         // Done, Aborted or Error ?
         IF (_response.State >= CmdMessageState.DONE )
         THEN
           // Rest Busy flag
           Busy := FALSE;
           // Update results
           OutCmd.LoadData          := _response.LoadData;
           OutCmd.LoadDataAvailable := _response.LoadDataAvailable;
           // set timeout
           SetTimeout(PT := _timeoutCmd, rTimer := _timerCmd);
           // inc step counter
          _stepCmd := _stepCmd + 1; 
         END_IF
       END_IF


  02: IF ( NOT Execute)
      THEN
        Reset();
      END_IF     

ELSE
  // invalid step
  ErrorID := RobotLibraryEvents.ERR_INVALID_STEP;
END_CASE


// Reset FB
IF ( NOT Execute )
THEN
  Reset();  
END_IF
END_METHOD

METHOD INTERNAL ParseResponsePayload : DINT
VAR_INPUT
  /// Response data
  ResponseData : RobotLibraryRecvDataFB;
  /// Timestamp
  Timestamp    : SystemTime;  
END_VAR
// Table 6-785: Received CMD payload (RC to PLC) of "LoadMeasurementSequential"
// --------------------------
// Header
// --------------------------
// Byte 00 : USINT - ParSeq | State     
// Byte 01 : SINT  - AlarmMessageSeverity    
// Byte 02 : UINT  - AlarmMessageCode HB
// Byte 03 :       - AlarmMessageCode LB
// Datablock
// --------------------------
// Byte 004 : IEC_DATE   - IEC Date LW HB
// Byte 005 :            - IEC Date LW LB
// Byte 006 : IEC_TIME   - IEC Time HW HB
// Byte 007 :            - IEC Time HW LB
// Byte 008 :            - IEC Time LW HB
// Byte 009 :            - IEC Time LW LB
// Byte 010 : REAL       - LoadData.X HW HB
// Byte 011 :            - LoadData.X HW LB
// Byte 012 :            - LoadData.X LW HB
// Byte 013 :            - LoadData.X LW LB
// Byte 014 : REAL       - LoadData.Y HW HB
// Byte 015 :            - LoadData.Y HW LB
// Byte 016 :            - LoadData.Y LW HB
// Byte 017 :            - LoadData.Y LW LB
// Byte 018 : REAL       - LoadData.Z HW HB
// Byte 019 :            - LoadData.Z HW LB
// Byte 020 :            - LoadData.Z LW HB
// Byte 021 :            - LoadData.Z LW LB
// Byte 022 : REAL       - LoadData.Rx HW HB
// Byte 023 :            - LoadData.Rx HW LB
// Byte 024 :            - LoadData.Rx LW HB
// Byte 025 :            - LoadData.Rx LW LB
// Byte 026 : REAL       - LoadData.Ry HW HB
// Byte 027 :            - LoadData.Ry HW LB
// Byte 028 :            - LoadData.Ry LW HB
// Byte 029 :            - LoadData.Ry LW LB
// Byte 030 : REAL       - LoadData.Rz HW HB
// Byte 031 :            - LoadData.Rz HW LB
// Byte 032 :            - LoadData.Rz LW HB
// Byte 033 :            - LoadData.Rz LW LB
// Byte 034 : REAL       - Mass HW HB
// Byte 035 :            - Mass HW LB
// Byte 036 :            - Mass LW HB
// Byte 037 :            - Mass LW LB
// Byte 038 : REAL       - LoadData.Ix HW HB
// Byte 039 :            - LoadData.Ix HW LB
// Byte 040 :            - LoadData.Ix LW HB
// Byte 041 :            - LoadData.Ix LW LB
// Byte 042 : REAL       - LoadData.Iy HW HB
// Byte 043 :            - LoadData.Iy HW LB
// Byte 044 :            - LoadData.Iy LW HB
// Byte 045 :            - LoadData.Iy LW LB
// Byte 046 : REAL       - LoadData.Iz HW HB
// Byte 047 :            - LoadData.Iz HW LB
// Byte 048 :            - LoadData.Iz LW HB
// Byte 049 :            - LoadData.Iz LW LB
// Byte 050 : BOOL       - LoadData.Available
// call base implementation to parse the header from payload buffer
ResponseData.PayloadPtr := SUPER^.ParseResponsePayload(ResponseData := ResponseData, Timestamp := Timestamp);

// copy parsed header to response
_response.ParSeq               := _rspHeader.ParSeq;
_response.State                := _rspHeader.State;
_response.AlarmMessageSeverity := _rspHeader.AlarmMessageSeverity;
_response.AlarmMessageCode     := _rspHeader.AlarmMessageCode;

// Get Response.LoadData.Timestamp.TsData
_response.LoadData.Timestamp.IEC_DATE := ResponseData.GetIecDate();
// Get Response.LoadData.Timestamp.TsTime
_response.LoadData.Timestamp.IEC_TIME := ResponseData.GetIecTime();
// Get Response.LoadData.X
_response.LoadData.X := ResponseData.GetReal();
// Get Response.LoadData.Y
_response.LoadData.Y := ResponseData.GetReal();
// Get Response.LoadData.Z
_response.LoadData.Z := ResponseData.GetReal();
// Get Response.LoadData.Rx
_response.LoadData.Rx := ResponseData.GetReal();
// Get Response.LoadData.Ry
_response.LoadData.Ry := ResponseData.GetReal();
// Get Response.LoadData.Rz
_response.LoadData.Rz := ResponseData.GetReal();
// Get Response.LoadData.Mass
_response.LoadData.Mass := ResponseData.GetReal();
// Get Response.LoadData.Ix
_response.LoadData.Ix := ResponseData.GetReal();
// Get Response.LoadData.Iy
_response.LoadData.Iy := ResponseData.GetReal();
// Get Response.LoadData.Iz
_response.LoadData.Iz := ResponseData.GetReal();
// Get Response.LoadDataAvailable
_response.LoadDataAvailable := ResponseData.GetBool();

// Create logging
ParseResponsePayloadLog(ResponseData := ResponseData, Timestamp := Timestamp);
END_METHOD

METHOD INTERNAL ParseResponsePayloadLog
VAR_INPUT
  /// Response data
  ResponseData : RobotLibraryRecvDataFB;
  /// Timestamp
  Timestamp    : SystemTime;  
END_VAR
// Create log entry for Parameter start
CreateLogMessage      ( Timestamp   := Timestamp,
                        MessageType := MessageType.CMD,
                        Severity    := Severity.DEBUG,
                        MessageCode := 0,
                        MessageText := 'Parsed the following parameter(s) from response data:');
                        
// Create log entry for LoadData.Timestamp.IEC_DATE
CreateLogMessagePara1 ( Timestamp   := Timestamp,
                        MessageType := MessageType.CMD,
                        Severity    := Severity.DEBUG,
                        MessageCode := 0,
                        MessageText := 'Response.LoadData.Timestamp.IEC_DATE = {1}',
                        Para1       :=  IEC_DATE_TO_STRING(_response.LoadData.Timestamp.IEC_DATE));

// Create log entry for LoadData.Timestamp.IEC_TIME
CreateLogMessagePara1 ( Timestamp   := Timestamp,
                        MessageType := MessageType.CMD,
                        Severity    := Severity.DEBUG,
                        MessageCode := 0,
                        MessageText := 'Response.LoadData.Timestamp.IEC_TIME = {1}',
                        Para1       :=  IEC_TIME_TO_STRING(_response.LoadData.Timestamp.IEC_TIME));

// Create log entry for LoadData.X
CreateLogMessagePara1 ( Timestamp   := Timestamp,
                        MessageType := MessageType.CMD,
                        Severity    := Severity.DEBUG,
                        MessageCode := 0,
                        MessageText := 'Response.LoadData.X = {1}',
                        Para1       :=  REAL_TO_STRING(_response.LoadData.X));

// Create log entry for LoadData.Y
CreateLogMessagePara1 ( Timestamp   := Timestamp,
                        MessageType := MessageType.CMD,
                        Severity    := Severity.DEBUG,
                        MessageCode := 0,
                        MessageText := 'Response.LoadData.Y = {1}',
                        Para1       :=  REAL_TO_STRING(_response.LoadData.Y));

// Create log entry for LoadData.Z
CreateLogMessagePara1 ( Timestamp   := Timestamp,
                        MessageType := MessageType.CMD,
                        Severity    := Severity.DEBUG,
                        MessageCode := 0,
                        MessageText := 'Response.LoadData.Z = {1}',
                        Para1       :=  REAL_TO_STRING(_response.LoadData.Z));

// Create log entry for LoadData.Rx
CreateLogMessagePara1 ( Timestamp   := Timestamp,
                        MessageType := MessageType.CMD,
                        Severity    := Severity.DEBUG,
                        MessageCode := 0,
                        MessageText := 'Response.LoadData.Rx = {1}',
                        Para1       :=  REAL_TO_STRING(_response.LoadData.Rx));

// Create log entry for LoadData.Ry
CreateLogMessagePara1 ( Timestamp   := Timestamp,
                        MessageType := MessageType.CMD,
                        Severity    := Severity.DEBUG,
                        MessageCode := 0,
                        MessageText := 'Response.LoadData.Ry = {1}',
                        Para1       :=  REAL_TO_STRING(_response.LoadData.Ry));

// Create log entry for LoadData.Rz
CreateLogMessagePara1 ( Timestamp   := Timestamp,
                        MessageType := MessageType.CMD,
                        Severity    := Severity.DEBUG,
                        MessageCode := 0,
                        MessageText := 'Response.LoadData.Rz = {1}',
                        Para1       :=  REAL_TO_STRING(_response.LoadData.Rz));

// Create log entry for LoadData.Mass
CreateLogMessagePara1 ( Timestamp   := Timestamp,
                        MessageType := MessageType.CMD,
                        Severity    := Severity.DEBUG,
                        MessageCode := 0,
                        MessageText := 'Response.LoadData.Mass = {1}',
                        Para1       :=  REAL_TO_STRING(_response.LoadData.Mass));

// Create log entry for LoadData.Ix
CreateLogMessagePara1 ( Timestamp   := Timestamp,
                        MessageType := MessageType.CMD,
                        Severity    := Severity.DEBUG,
                        MessageCode := 0,
                        MessageText := 'Response.LoadData.Ix = {1}',
                        Para1       :=  REAL_TO_STRING(_response.LoadData.Ix));

// Create log entry for LoadData.Iy
CreateLogMessagePara1 ( Timestamp   := Timestamp,
                        MessageType := MessageType.CMD,
                        Severity    := Severity.DEBUG,
                        MessageCode := 0,
                        MessageText := 'Response.LoadData.Iy = {1}',
                        Para1       :=  REAL_TO_STRING(_response.LoadData.Iy));

// Create log entry for LoadData.Iz
CreateLogMessagePara1 ( Timestamp   := Timestamp,
                        MessageType := MessageType.CMD,
                        Severity    := Severity.DEBUG,
                        MessageCode := 0,
                        MessageText := 'Response.LoadData.Iz = {1}',
                        Para1       :=  REAL_TO_STRING(_response.LoadData.Iz));

// Create log entry for LoadDataAvailable
CreateLogMessagePara1 ( Timestamp   := Timestamp,
                        MessageType := MessageType.CMD,
                        Severity    := Severity.DEBUG,
                        MessageCode := 0,
                        MessageText := 'Response.LoadDataAvailable = {1}',
                        Para1       :=  BOOL_TO_STRING(_response.LoadDataAvailable));
END_METHOD

METHOD PROTECTED Reset : DINT
VAR_INPUT
END_VAR
Reset := SUPER^.Reset();

Done               := FALSE;
Busy               := FALSE;
Active             := FALSE;
CommandBuffered    := FALSE;
CommandAborted     := FALSE;
CommandInterrupted := FALSE;
END_METHOD

END_FUNCTION_BLOCK

// Library/POUs/ConveyorTracking/MC_ActivateConveyorTracking/MC_ActivateConveyorTrackingFB
/// Activate conveyor tracking mode
FUNCTION_BLOCK MC_ActivateConveyorTrackingFB EXTENDS RobotLibraryBaseFB
// ------------------------------------------------------------------------- 
//  SRCI Robot Library                                                
// ------------------------------------------------------------------------- 
//                                                                           
//  Object:      ActivateConveyorTrackingFB                                       
//  Author:      Thorsten Brach                                                
//  Date:        2024-06-11
//
//  Description:                                              
//   
//                                                                           
//  Copyright: 
//    (C) 2024 Thorsten Brach. All rights reserved                                                                                                                                            
//             Licensed under the LGPL-3.0 license.
//                                                                           
//  Disclaimer:                                                                           
//    This project is provided without any guarantee and can be used for   
//    private and commercial purposes. Any use is at the user’s 
//    own risk and responsibility.
//
// -------------------------------------------------------------------------
VAR_INPUT
  /// SSet TRUE to activate conveyor tracking functionality
  Enable             : BOOL;
  /// Command parameter 
  ParCmd             : ActivateConveyorTrackingParCmd;      
END_VAR

VAR_OUTPUT
  /// TRUE, while the following outputs return valid values:
  /// • TrackingStatusByte
  /// • RCEncoderValue
  Valid              : BOOL;
  /// FB is being processed
  Busy               : BOOL;
  /// Command is transferred and confirmed by the RC
  CommandBuffered    : BOOL;
  /// Receiving of input parameter values has been acknowledged by RC
  ParameterAccepted  : BOOL;
  /// Command output 
  OutCmd             : ActivateConveyorTrackingOutCmd;  
END_VAR

VAR
  /// internal copy of command parameter 
 _parCmd             : ActivateConveyorTrackingParCmd;
  /// command data to send
 _command            : ActivateConveyorTrackingSendData;
  /// response data received
 _response           : ActivateConveyorTrackingRecvData;  
  /// Rising edge for enable
 _enable_R          : R_TRIG;
  /// Falling edge for enable
 _enable_F          : F_TRIG;    
END_VAR

SUPER^(AxesGroup := AxesGroup);

METHOD PROTECTED CheckFunctionSupported : BOOL
VAR_IN_OUT
  /// Robot assignment of function
  AxesGroup : AxesGroup; 
END_VAR
CheckFunctionSupported := AxesGroup.InternalData.RCSupportedFunctions.ActivateConveyorTracking;

IF ( NOT CheckFunctionSupported )
THEN
  // call base implementation for set error and create log entry
  SUPER^.CheckFunctionSupported(AxesGroup := AxesGroup);
END_IF
END_METHOD

METHOD PROTECTED CheckParameterChanged : BOOL
VAR_IN_OUT
  /// Robot assignment of function
  AxesGroup    : AxesGroup; 
END_VAR
// Check ParCmd Size is > 0, because MemCmp does not work correctly with size = 0
IF (SIZEOF(ParCmd) = 0) 
THEN 
  RETURN;
END_IF

// compare memory 
_parameterChanged := ( SysDepMemCmp(pData1 := ADR(ParCmd), pData2 := ADR(_parCmd), DataLen := SIZEOF(ParCmd)) <> RobotLibraryConstants.OK );

// check parameter valid ?
_parameterValid   := CheckParameterValid( AxesGroup := AxesGroup );

IF ((  _parameterChanged        )  AND 
    (  _parameterValid          )) OR
    (  _parameterUpdateInternal )  
THEN  
  // reset internal flag for send parameter update
 _parameterUpdateInternal := FALSE;
  // update internal copy of parameters 
 _parCmd := ParCmd;
  // inc parameter sequence
 _command.ParSeq := _command.ParSeq + 1;
  // update command data  
  CommandData := CreateCommandPayload(AxesGroup := AxesGroup); // ( Access via reference to rCommandFB in ACR )
  // notify active command register 
  AxesGroup.Acyclic.ActiveCommandRegister.NotifyParameterChanged := _uniqueID;
  // Reset parameter accepted flag
  ParameterAccepted := FALSE;  
END_IF
END_METHOD

METHOD INTERNAL CreateCommandPayload : RobotLibrarySendDataFB
VAR_IN_OUT
  /// Robot assignment of function
  AxesGroup : AxesGroup; 
END_VAR
// Table 6-438: Sent CMD payload (PLC to RC) of "ActivateConveyorTracking"
// --------------------------
// Header
// --------------------------
// Byte 00 : UINT  - Type HB     
// Byte 01 :       - Type LB    
// Byte 02 : USINT - Reserve | ExecutionMode
// Byte 03 : USINT - ParSeq  | Priority
// --------------------------
// Datablock
// --------------------------
// Byte 04 : SINT  - ConveyorNo
// Byte 05 : SINT  - ConnectionMode
// --------------------------


// set command parameter 
_command.CmdTyp         :=  CmdType.ActivateConveyorTracking;
_command.ExecMode       :=  ExecMode;
_command.ParSeq         := _command.ParSeq;
_command.Priority       :=  Priority;
_command.ConveyorNo     := _parCmd.ConveyorNo;
_command.ConnectionMode := _parCmd.ConnectionMode;


// copy command data to header
_cmdHeader := _command;
// call base implementation to copy header to payload buffer
CreateCommandPayload := SUPER^.CreateCommandPayload(AxesGroup := AxesGroup);


// add command.ConveyorNo
CreateCommandPayload.AddSint(_command.ConveyorNo);
// add command.ConnectionMode
CreateCommandPayload.AddSint(_command.ConnectionMode);

// Create logging
CreateCommandPayloadLog(AxesGroup := AxesGroup);
END_METHOD

METHOD INTERNAL CreateCommandPayloadLog 
VAR_IN_OUT
  /// Robot assignment of function
  AxesGroup : AxesGroup; 
END_VAR
// Create log entry for Parameter start
CreateLogMessage      ( Timestamp   := AxesGroup.InternalData.SystemTime,
                        MessageType := MessageType.CMD,
                        Severity    := Severity.DEBUG,
                        MessageCode := 0,
                        MessageText := 'Create command payload with the following parameter(s) :');

// Create log entry for ConveyorNo
CreateLogMessagePara1 ( Timestamp   := AxesGroup.InternalData.SystemTime,
                        MessageType := MessageType.CMD,
                        Severity    := Severity.DEBUG,
                        MessageCode := 0,
                        MessageText := 'Command.ConveyorNo = {1}',
                        Para1       :=  SINT_TO_STRING(_command.ConveyorNo));
                        
// Create log entry for ConnectionMode
CreateLogMessagePara1 ( Timestamp   := AxesGroup.InternalData.SystemTime,
                        MessageType := MessageType.CMD,
                        Severity    := Severity.DEBUG,
                        MessageCode := 0,
                        MessageText := 'Command.ConnectionMode = {1}',
                        Para1       :=  CONNECTION_MODE_TO_STRING(_command.ConnectionMode));
END_METHOD

METHOD FB_init : BOOL
VAR_INPUT
  /// if TRUE, the retain variables are initialized (warm start / cold start)
  bInitRetains : BOOL; 
  /// if TRUE, the instance afterwards gets moved into the copy code (online change)
  bInCopyCode  : BOOL;  
END_VAR
MyType := 'MC_ActivateConveyorTrackingFB';
END_METHOD

METHOD PROTECTED OnCall
VAR_IN_OUT
  /// Robot assignment of function
  AxesGroup : AxesGroup; 
END_VAR
// call base implementation
SUPER^.OnCall(AxesGroup := AxesGroup);

// building rising and falling edges
_enable_R( CLK := Enable);
_enable_F( CLK := Enable);

CASE _stepCmd OF
  
  00:  IF ( _enable_R.Q ) 
       THEN
         // reset the rising edge
        _enable_R();       
         // reset the falling edge
        _enable_F();       

         // Check function is supported and parameter are valid ?
         IF (( CheckFunctionSupported( AxesGroup := AxesGroup )) AND
             ( CheckParameterValid   ( AxesGroup := AxesGroup )))      
         THEN
           // set busy flag
           Busy := TRUE;
           // Reset command outputs
           SysDepMemSet(pDest := ADR(OutCmd), Value := 0, DataLen := SIZEOF(OutCmd));         
           // apply command parameter
          _parCmd := ParCmd;
           // init parameter sequence
          _command.ParSeq := 1;
           // create command data
           CommandData := CreateCommandPayload(AxesGroup := AxesGroup);
           // Add command to active command register
          _uniqueID := AxesGroup.Acyclic.ActiveCommandRegister.AddCmd( pCommandFB := ADR(THIS^ ));     
           // set timeout
           SetTimeout(PT := _timeoutCmd, rTimer := _timerCmd);
           // inc step counter
          _stepCmd := _stepCmd + 1;
         END_IF 
       END_IF
     

  01:  // Wait for responce received
       IF ( _responseReceived )
       THEN
         // reset response received flag
        _responseReceived := FALSE;

         CASE  _response.State 
         OF
           CmdMessageState.BUFFERED    : CommandBuffered    := TRUE;
           CmdMessageState.ACTIVE      : ParameterAccepted  := TRUE;           
           CmdMessageState.ERROR       : Error              := TRUE;
         END_CASE
                
         // Done, Aborted or Error ?
         IF (_response.State >= CmdMessageState.DONE )
         THEN
           // Update results
           OutCmd.TrackingStatus := _response.TrackingStatus;
           // set timeout
           SetTimeout(PT := _timeoutCmd, rTimer := _timerCmd);
           // inc step counter
          _stepCmd := _stepCmd + 1; 
         END_IF
       END_IF


  02: IF (NOT Enable)
      THEN
        Reset();
	    END_IF
      
ELSE
  // invalid step
  ErrorID := RobotLibraryEvents.ERR_INVALID_STEP;
END_CASE



// Reset FB
IF (( _enable_R.Q ) OR
    ( _enable_F.Q ))
THEN
  Reset();
END_IF
END_METHOD

METHOD INTERNAL ParseResponsePayload : DINT
VAR_INPUT
  /// Response data
  ResponseData : RobotLibraryRecvDataFB;
  /// Timestamp
  Timestamp    : SystemTime;  
END_VAR
// Table 6-439: Received CMD payload (RC to PLC) of "ActivateConveyorTracking"
// --------------------------
// Header
// --------------------------
// Byte 00 : USINT - ParSeq | State     
// Byte 01 : SINT  - AlarmMessageSeverity    
// Byte 02 : UINT  - AlarmMessageCode HB
// Byte 03 :       - AlarmMessageCode LB
// --------------------------
// Datablock
// --------------------------
// Byte 04 : BYTE  - TrackingStatusByte
// --------------------------
// call base implementation to parse the header from payload buffer
ResponseData.PayloadPtr := SUPER^.ParseResponsePayload(ResponseData := ResponseData, Timestamp := Timestamp);

// copy parsed header to response
_response.ParSeq               := _rspHeader.ParSeq;
_response.State                := _rspHeader.State;
_response.AlarmMessageSeverity := _rspHeader.AlarmMessageSeverity;
_response.AlarmMessageCode     := _rspHeader.AlarmMessageCode;

// Get Response.Enabled
_response.TrackingStatus := ResponseData.GetTrackingStatus();

// Create logging
ParseResponsePayloadLog(ResponseData := ResponseData, Timestamp := Timestamp);
END_METHOD

METHOD INTERNAL ParseResponsePayloadLog
VAR_INPUT
  /// Response data
  ResponseData : RobotLibraryRecvDataFB;
  /// Timestamp
  Timestamp    : SystemTime;  
END_VAR
// Create log entry for Parameter start
CreateLogMessage      ( Timestamp   := Timestamp,
                        MessageType := MessageType.CMD,
                        Severity    := Severity.DEBUG,
                        MessageCode := 0,
                        MessageText := 'Parsed the following parameter(s) from response data:');
                        
// Create log entry for TrackingStatus.ConveyorTrackingEnabled
CreateLogMessagePara1 ( Timestamp   := Timestamp,
                        MessageType := MessageType.CMD,
                        Severity    := Severity.DEBUG,
                        MessageCode := 0,
                        MessageText := 'Response.TrackingStatus.ConveyorTrackingEnabled = {1}',
                        Para1       :=  BOOL_TO_STRING(_response.TrackingStatus.ConveyorTrackingEnabled));

// Create log entry for TrackingStatus.WaitingForSynchronization
CreateLogMessagePara1 ( Timestamp   := Timestamp,
                        MessageType := MessageType.CMD,
                        Severity    := Severity.DEBUG,
                        MessageCode := 0,
                        MessageText := 'Response.TrackingStatus.WaitingForSynchronization = {1}',
                        Para1       :=  BOOL_TO_STRING(_response.TrackingStatus.WaitingForSynchronization));

// Create log entry for TrackingStatus.Synchronizing
CreateLogMessagePara1 ( Timestamp   := Timestamp,
                        MessageType := MessageType.CMD,
                        Severity    := Severity.DEBUG,
                        MessageCode := 0,
                        MessageText := 'Response.TrackingStatus.Synchronizing = {1}',
                        Para1       :=  BOOL_TO_STRING(_response.TrackingStatus.Synchronizing));

// Create log entry for TrackingStatus.Synchronous
CreateLogMessagePara1 ( Timestamp   := Timestamp,
                        MessageType := MessageType.CMD,
                        Severity    := Severity.DEBUG,
                        MessageCode := 0,
                        MessageText := 'Response.TrackingStatus.Synchronous = {1}',
                        Para1       :=  BOOL_TO_STRING(_response.TrackingStatus.Synchronous));

// Create log entry for TrackingStatus.Desynchronizing
CreateLogMessagePara1 ( Timestamp   := Timestamp,
                        MessageType := MessageType.CMD,
                        Severity    := Severity.DEBUG,
                        MessageCode := 0,
                        MessageText := 'Response.TrackingStatus.Desynchronizing = {1}',
                        Para1       :=  BOOL_TO_STRING(_response.TrackingStatus.Desynchronizing));

// Create log entry for TrackingStatus.SyncOutZoneEntered
CreateLogMessagePara1 ( Timestamp   := Timestamp,
                        MessageType := MessageType.CMD,
                        Severity    := Severity.DEBUG,
                        MessageCode := 0,
                        MessageText := 'Response.TrackingStatus.SyncOutZoneEntered = {1}',
                        Para1       :=  BOOL_TO_STRING(_response.TrackingStatus.SyncOutZoneEntered));

// Create log entry for TrackingStatus.SyncOutZoneLeft
CreateLogMessagePara1 ( Timestamp   := Timestamp,
                        MessageType := MessageType.CMD,
                        Severity    := Severity.DEBUG,
                        MessageCode := 0,
                        MessageText := 'Response.TrackingStatus.SyncOutZoneLeft = {1}',
                        Para1       :=  BOOL_TO_STRING(_response.TrackingStatus.SyncOutZoneLeft));

// Create log entry for TrackingStatus.NotUsed
CreateLogMessagePara1 ( Timestamp   := Timestamp,
                        MessageType := MessageType.CMD,
                        Severity    := Severity.DEBUG,
                        MessageCode := 0,
                        MessageText := 'Response.TrackingStatus.NotUsed = {1}',
                        Para1       :=  BOOL_TO_STRING(_response.TrackingStatus.NotUsed));
END_METHOD

METHOD PROTECTED Reset : DINT
VAR_INPUT
END_VAR
Reset := SUPER^.Reset();

Valid              := FALSE;
Busy               := FALSE;
CommandBuffered    := FALSE;
ParameterAccepted  := FALSE;
END_METHOD

END_FUNCTION_BLOCK

// Library/POUs/ConveyorTracking/MC_ConfigureConveyor/MC_ConfigureConveyorFB
/// Configure conveyor parameters
FUNCTION_BLOCK MC_ConfigureConveyorFB EXTENDS RobotLibraryBaseExecuteFB
// ------------------------------------------------------------------------- 
//  SRCI Robot Library                                                
// ------------------------------------------------------------------------- 
//                                                                           
//  Object:      ConfigureConveyorFB                                       
//  Author:      Thorsten Brach                                                
//  Date:        2024-06-11
//
//  Description:                                              
//   
//                                                                           
//  Copyright: 
//    (C) 2024 Thorsten Brach. All rights reserved                                                                                                                                            
//             Licensed under the LGPL-3.0 license.
//                                                                           
//  Disclaimer:                                                                           
//    This project is provided without any guarantee and can be used for   
//    private and commercial purposes. Any use is at the user’s 
//    own risk and responsibility.
//
// -------------------------------------------------------------------------
VAR_INPUT
  /// Command parameter 
  ParCmd          : ConfigureConveyorParCmd;      
END_VAR

VAR_OUTPUT
  /// Command is transferred and confirmed by the RC
  CommandBuffered : BOOL;
  /// Command output 
  OutCmd          : ConfigureConveyorOutCmd;  
END_VAR

VAR
  /// internal copy of command parameter 
 _parCmd          : ConfigureConveyorParCmd;
  /// command data to send
 _command         : ConfigureConveyorSendData;
  /// response data received
 _response        : ConfigureConveyorRecvData;      
END_VAR

SUPER^(AxesGroup := AxesGroup);

METHOD PROTECTED CheckFunctionSupported : BOOL
VAR_IN_OUT
  /// Robot assignment of function
  AxesGroup : AxesGroup; 
END_VAR
CheckFunctionSupported := AxesGroup.InternalData.RCSupportedFunctions.ConfigureConveyor;

IF ( NOT CheckFunctionSupported )
THEN
  // call base implementation for set error and create log entry
  SUPER^.CheckFunctionSupported(AxesGroup := AxesGroup);
END_IF
END_METHOD

METHOD PROTECTED CheckParameterChanged : BOOL
VAR_IN_OUT
  /// Robot assignment of function
  AxesGroup    : AxesGroup; 
END_VAR
// Check ParCmd Size is > 0, because MemCmp does not work correctly with size = 0
IF (SIZEOF(ParCmd) = 0) 
THEN 
  RETURN;
END_IF

// compare memory 
_parameterChanged := ( SysDepMemCmp(pData1 := ADR(ParCmd), pData2 := ADR(_parCmd), DataLen := SIZEOF(ParCmd)) <> RobotLibraryConstants.OK );

// check parameter valid ?
_parameterValid   := CheckParameterValid( AxesGroup := AxesGroup );

IF ((  _parameterChanged        )  AND 
    (  _parameterValid          )) OR
    (  _parameterUpdateInternal )  
THEN  
  // reset internal flag for send parameter update
 _parameterUpdateInternal := FALSE;
  // update internal copy of parameters 
 _parCmd := ParCmd;
  // inc parameter sequence
 _command.ParSeq := _command.ParSeq + 1;
  // update command data  
  CommandData := CreateCommandPayload(AxesGroup := AxesGroup); // ( Access via reference to rCommandFB in ACR )
  // notify active command register 
  AxesGroup.Acyclic.ActiveCommandRegister.NotifyParameterChanged := _uniqueID;
END_IF
END_METHOD

METHOD INTERNAL CreateCommandPayload : RobotLibrarySendDataFB
VAR_IN_OUT
  /// Robot assignment of function
  AxesGroup : AxesGroup; 
END_VAR
// Table 6-458: Sent CMD payload (PLC to RC) of "ConfigureConveyor"
// --------------------------
// Header
// --------------------------
// Byte 00 : UINT       - Type HB     
// Byte 01 :            - Type LB    
// Byte 02 : USINT      - Reserve | ExecutionMode
// Byte 03 : USINT      - ParSeq  | Priority
// --------------------------
// Datablock
// --------------------------
// Byte 04 : IEC_DATE   - Date              LW HB
// Byte 05 :            - Date              LW LB
// Byte 06 : IEC_TIME   - Time              HW HB
// Byte 07 :            - Time              HW LB
// Byte 08 :            - Time              LW HB
// Byte 09 :            - Time              LW LB
// Byte 10 : USINT      - ReferenceFrame
// Byte 11 : BYTE       - Reserve
// Byte 12 : REAL       - ConveyorOrigin.X  HW HB
// Byte 13 :            - ConveyorOrigin.X  HW LB
// Byte 14 :            - ConveyorOrigin.X  LW HB
// Byte 15 :            - ConveyorOrigin.X  LW LB
// Byte 16 : REAL       - ConveyorOrigin.Y  HW HB
// Byte 17 :            - ConveyorOrigin.Y  HW LB
// Byte 18 :            - ConveyorOrigin.Y  LW HB
// Byte 19 :            - ConveyorOrigin.Y  LW LB
// Byte 20 : REAL       - ConveyorOrigin.Z  HW HB
// Byte 21 :            - ConveyorOrigin.Z  HW LB
// Byte 22 :            - ConveyorOrigin.Z  LW HB
// Byte 23 :            - ConveyorOrigin.Z  LW LB
// Byte 24 : REAL       - ConveyorOrigin.Rx HW HB
// Byte 25 :            - ConveyorOrigin.Rx HW LB
// Byte 26 :            - ConveyorOrigin.Rx LW HB
// Byte 27 :            - ConveyorOrigin.Rx LW LB
// Byte 28 : REAL       - ConveyorOrigin.Ry HW HB
// Byte 29 :            - ConveyorOrigin.Ry HW LB
// Byte 30 :            - ConveyorOrigin.Ry LW HB
// Byte 31 :            - ConveyorOrigin.Ry LW LB
// Byte 32 : REAL       - ConveyorOrigin.Rz HW HB
// Byte 33 :            - ConveyorOrigin.Rz HW LB
// Byte 34 :            - ConveyorOrigin.Rz LW HB
// Byte 35 :            - ConveyorOrigin.Rz LW LB
// Byte 36 : BOOL       - ConveyorOrigin Available
// Byte 37 : USINT      - ConveyorNo
// Byte 38 : USINT      - ConveyorType
// Byte 39 : REAL       - Radius            HW HB
// Byte 40 :            - Radius            HW LB
// Byte 41 :            - Radius            LW HB
// Byte 42 :            - Radius            LW LB
// Byte 43 : REAL       - StartDistance     HW HB
// Byte 44 :            - StartDistance     HW LB
// Byte 45 :            - StartDistance     LW HB
// Byte 46 :            - StartDistance     LW LB
// Byte 47 : REAL       - EndDistance       HW HB
// Byte 48 :            - EndDistance       HW LB
// Byte 49 :            - EndDistance       LW HB
// Byte 50 :            - EndDistance       LW LB
// Byte 51 : REAL       - SyncInLength      HW HB
// Byte 52 :            - SyncInLength      HW LB
// Byte 53 :            - SyncInLength      LW HB
// Byte 54 :            - SyncInLength      LW LB
// Byte 55 : REAL       - SyncOutLength     HW HB
// Byte 56 :            - SyncOutLength     HW LB
// Byte 57 :            - SyncOutLength     LW HB
// Byte 58 :            - SyncOutLength     LW LB
// --------------------------
// set command parameter 
_command.CmdTyp         :=  CmdType.ConfigureConveyor;
_command.ExecMode       :=  ExecMode;
_command.ParSeq         := _command.ParSeq;
_command.Priority       :=  Priority;
_command.ConveyorNo     := _parCmd.ConveyorNo;
_command.ConveyorOrigin := _parCmd.ConveyorOrigin;
_command.ConveyorType   := _parCmd.ConveyorType;
_command.Radius         := _parCmd.Radius;
_command.StartDistance  := _parCmd.StartDistance;
_command.EndDistance    := _parCmd.EndDistance;
_command.SyncInLength   := _parCmd.SyncInLength;
_command.SyncOutLength  := _parCmd.SyncOutLength;

// copy command data to header
_cmdHeader := _command;
// call base implementation to copy header to payload buffer
CreateCommandPayload := SUPER^.CreateCommandPayload(AxesGroup := AxesGroup);


// add command.ConveyorOrigin.Timestamp.IEC_DATE
CreateCommandPayload.AddIecDate(_command.ConveyorOrigin.Timestamp.IEC_DATE);
// add command.ConveyorOrigin.Timestamp.IEC_TIME
CreateCommandPayload.AddIecTime(_command.ConveyorOrigin.Timestamp.IEC_TIME);
// add command.ConveyorOrigin.ReferenceFrame
CreateCommandPayload.AddUsint(_command.ConveyorOrigin.ReferenceFrame);
// add command.ConveyorOrigin.Reserve
CreateCommandPayload.AddByte(0);
// add command.ConveyorOrigin.ReferenceFrame.X
CreateCommandPayload.AddReal(_command.ConveyorOrigin.X);
// add command.ConveyorOrigin.ReferenceFrame.Y
CreateCommandPayload.AddReal(_command.ConveyorOrigin.Y);
// add command.ConveyorOrigin.ReferenceFrame.Z
CreateCommandPayload.AddReal(_command.ConveyorOrigin.Z);
// add command.ConveyorOrigin.ReferenceFrame.Rx
CreateCommandPayload.AddReal(_command.ConveyorOrigin.Rx);
// add command.ConveyorOrigin.ReferenceFrame.Ry
CreateCommandPayload.AddReal(_command.ConveyorOrigin.Ry);
// add command.ConveyorOrigin.ReferenceFrame.Rz
CreateCommandPayload.AddReal(_command.ConveyorOrigin.Rz);
// add command.ConveyorOriginAvailable
CreateCommandPayload.AddBool(_command.ConveyorOriginAvailable);
// add command.ConveyorNo
CreateCommandPayload.AddUsint(_command.ConveyorNo);
// add command.ConveyorType
CreateCommandPayload.AddUsint(_command.ConveyorType);
// add command.Radius
CreateCommandPayload.AddReal(_command.Radius);
// add command.StartDistance
CreateCommandPayload.AddReal(_command.StartDistance);
// add command.EndDistance
CreateCommandPayload.AddReal(_command.EndDistance);
// add command.SyncInLength
CreateCommandPayload.AddReal(_command.SyncInLength);
// add command.SyncOutLength
CreateCommandPayload.AddReal(_command.SyncOutLength);

// Create logging
CreateCommandPayloadLog(AxesGroup := AxesGroup);
END_METHOD

METHOD INTERNAL CreateCommandPayloadLog 
VAR_IN_OUT
  /// Robot assignment of function
  AxesGroup : AxesGroup; 
END_VAR
// Create log entry for Parameter start
CreateLogMessage      ( Timestamp   := AxesGroup.InternalData.SystemTime,
                        MessageType := MessageType.CMD,
                        Severity    := Severity.DEBUG,
                        MessageCode := 0,
                        MessageText := 'Create command payload with the following parameter(s) :');

// Create log entry for ConveyorOrigin.Timestamp.IEC_DATE
CreateLogMessagePara1 ( Timestamp   := AxesGroup.InternalData.SystemTime,
                        MessageType := MessageType.CMD,
                        Severity    := Severity.DEBUG,
                        MessageCode := 0,
                        MessageText := 'Command.ConveyorOrigin.Timestamp.IEC_DATE = {1}',
                        Para1       :=  IEC_DATE_TO_STRING(_command.ConveyorOrigin.Timestamp.IEC_DATE));
                       
// Create log entry for ConveyorOrigin.Timestamp.IEC_TIME
CreateLogMessagePara1 ( Timestamp   := AxesGroup.InternalData.SystemTime,
                        MessageType := MessageType.CMD,
                        Severity    := Severity.DEBUG,
                        MessageCode := 0,
                        MessageText := 'Command.ConveyorOrigin.Timestamp.IEC_TIME = {1}',
                        Para1       :=  IEC_TIME_TO_STRING(_command.ConveyorOrigin.Timestamp.IEC_TIME));

// Create log entry for ConveyorOrigin.ReferenceFrame
CreateLogMessagePara1 ( Timestamp   := AxesGroup.InternalData.SystemTime,
                        MessageType := MessageType.CMD,
                        Severity    := Severity.DEBUG,
                        MessageCode := 0,
                        MessageText := 'Command.ConveyorOrigin.ReferenceFrame = {1}',
                        Para1       :=  USINT_TO_STRING(_command.ConveyorOrigin.ReferenceFrame));
                        
// Create log entry for Reserve
CreateLogMessagePara1 ( Timestamp   := AxesGroup.InternalData.SystemTime,
                        MessageType := MessageType.CMD,
                        Severity    := Severity.DEBUG,
                        MessageCode := 0,
                        MessageText := 'Command.Reserve = {1}',
                        Para1       :=  BYTE_TO_STRING(0));        

// Create log entry for ConveyorOrigin.X
CreateLogMessagePara1 ( Timestamp   := AxesGroup.InternalData.SystemTime,
                        MessageType := MessageType.CMD,
                        Severity    := Severity.DEBUG,
                        MessageCode := 0,
                        MessageText := 'Command.ConveyorOrigin.X = {1}',
                        Para1       :=  REAL_TO_STRING(_command.ConveyorOrigin.X));
                        
// Create log entry for ConveyorOrigin.Y
CreateLogMessagePara1 ( Timestamp   := AxesGroup.InternalData.SystemTime,
                        MessageType := MessageType.CMD,
                        Severity    := Severity.DEBUG,
                        MessageCode := 0,
                        MessageText := 'Command.ConveyorOrigin.Y = {1}',
                        Para1       :=  REAL_TO_STRING(_command.ConveyorOrigin.Y));
                        
// Create log entry for ConveyorOrigin.Z
CreateLogMessagePara1 ( Timestamp   := AxesGroup.InternalData.SystemTime,
                        MessageType := MessageType.CMD,
                        Severity    := Severity.DEBUG,
                        MessageCode := 0,
                        MessageText := 'Command.ConveyorOrigin.Z = {1}',
                        Para1       :=  REAL_TO_STRING(_command.ConveyorOrigin.Z));

// Create log entry for ConveyorOrigin.Rx
CreateLogMessagePara1 ( Timestamp   := AxesGroup.InternalData.SystemTime,
                        MessageType := MessageType.CMD,
                        Severity    := Severity.DEBUG,
                        MessageCode := 0,
                        MessageText := 'Command.ConveyorOrigin.Rx = {1}',
                        Para1       :=  REAL_TO_STRING(_command.ConveyorOrigin.Rx));
                        
// Create log entry for ConveyorOrigin.Ry
CreateLogMessagePara1 ( Timestamp   := AxesGroup.InternalData.SystemTime,
                        MessageType := MessageType.CMD,
                        Severity    := Severity.DEBUG,
                        MessageCode := 0,
                        MessageText := 'Command.ConveyorOrigin.Ry = {1}',
                        Para1       :=  REAL_TO_STRING(_command.ConveyorOrigin.Ry));
                        
// Create log entry for ConveyorOrigin.Rz
CreateLogMessagePara1 ( Timestamp   := AxesGroup.InternalData.SystemTime,
                        MessageType := MessageType.CMD,
                        Severity    := Severity.DEBUG,
                        MessageCode := 0,
                        MessageText := 'Command.ConveyorOrigin.Rz = {1}',
                        Para1       :=  REAL_TO_STRING(_command.ConveyorOrigin.Rz));                        
                        
// Create log entry for ConveyorOriginAvailable
CreateLogMessagePara1 ( Timestamp   := AxesGroup.InternalData.SystemTime,
                        MessageType := MessageType.CMD,
                        Severity    := Severity.DEBUG,
                        MessageCode := 0,
                        MessageText := 'Command.ConveyorOriginAvailable = {1}',
                        Para1       :=  BOOL_TO_STRING(_command.ConveyorOriginAvailable));
                        
// Create log entry for ConveyorNo
CreateLogMessagePara1 ( Timestamp   := AxesGroup.InternalData.SystemTime,
                        MessageType := MessageType.CMD,
                        Severity    := Severity.DEBUG,
                        MessageCode := 0,
                        MessageText := 'Command.ConveyorNo = {1}',
                        Para1       :=  USINT_TO_STRING(_command.ConveyorNo));
                        
// Create log entry for ConveyorType
CreateLogMessagePara1 ( Timestamp   := AxesGroup.InternalData.SystemTime,
                        MessageType := MessageType.CMD,
                        Severity    := Severity.DEBUG,
                        MessageCode := 0,
                        MessageText := 'Command.ConveyorType = {1}',
                        Para1       :=  CONVEYOR_TYPE_TO_STRING(_command.ConveyorType));                        
                        
// Create log entry for Radius
CreateLogMessagePara1 ( Timestamp   := AxesGroup.InternalData.SystemTime,
                        MessageType := MessageType.CMD,
                        Severity    := Severity.DEBUG,
                        MessageCode := 0,
                        MessageText := 'Command.Radius = {1}',
                        Para1       :=  REAL_TO_STRING(_command.Radius));       
                        
// Create log entry for StartDistance
CreateLogMessagePara1 ( Timestamp   := AxesGroup.InternalData.SystemTime,
                        MessageType := MessageType.CMD,
                        Severity    := Severity.DEBUG,
                        MessageCode := 0,
                        MessageText := 'Command.StartDistance = {1}',
                        Para1       :=  REAL_TO_STRING(_command.StartDistance));       
    
// Create log entry for EndDistance
CreateLogMessagePara1 ( Timestamp   := AxesGroup.InternalData.SystemTime,
                        MessageType := MessageType.CMD,
                        Severity    := Severity.DEBUG,
                        MessageCode := 0,
                        MessageText := 'Command.EndDistance = {1}',
                        Para1       :=  REAL_TO_STRING(_command.EndDistance));           

// Create log entry for SyncInLength
CreateLogMessagePara1 ( Timestamp   := AxesGroup.InternalData.SystemTime,
                        MessageType := MessageType.CMD,
                        Severity    := Severity.DEBUG,
                        MessageCode := 0,
                        MessageText := 'Command.SyncInLength = {1}',
                        Para1       :=  REAL_TO_STRING(_command.SyncInLength));           

// Create log entry for SyncOutLength
CreateLogMessagePara1 ( Timestamp   := AxesGroup.InternalData.SystemTime,
                        MessageType := MessageType.CMD,
                        Severity    := Severity.DEBUG,
                        MessageCode := 0,
                        MessageText := 'Command.SyncOutLength = {1}',
                        Para1       :=  REAL_TO_STRING(_command.SyncOutLength));
END_METHOD

METHOD FB_init : BOOL
VAR_INPUT
  /// if TRUE, the retain variables are initialized (warm start / cold start)
  bInitRetains : BOOL; 
  /// if TRUE, the instance afterwards gets moved into the copy code (online change)
  bInCopyCode  : BOOL;  
END_VAR
MyType := 'MC_ConfigureConveyorFB';
END_METHOD

METHOD PROTECTED OnCall
VAR_IN_OUT
  /// Robot assignment of function
  AxesGroup : AxesGroup; 
END_VAR
// call base implementation
SUPER^.OnCall(AxesGroup := AxesGroup);

CASE _stepCmd OF
  
  00:  IF ( _execute_R.Q )  
       THEN
         // Check function is supported and parameter are valid ?
         IF (( CheckFunctionSupported( AxesGroup := AxesGroup )) AND
             ( CheckParameterValid   ( AxesGroup := AxesGroup )))      
         THEN
           // set busy flag
           Busy := TRUE;
           // Reset command outputs
           SysDepMemSet(pDest := ADR(OutCmd), Value := 0, DataLen := SIZEOF(OutCmd));         
           // apply command parameter
          _parCmd := ParCmd;
           // init parameter sequence
          _command.ParSeq := 1;
           // create command data
           CommandData := CreateCommandPayload(AxesGroup := AxesGroup);
           // Add command to active command register
          _uniqueID := AxesGroup.Acyclic.ActiveCommandRegister.AddCmd( pCommandFB := ADR(THIS^ ));     
           // set timeout
           SetTimeout(PT := _timeoutCmd, rTimer := _timerCmd);
           // inc step counter
          _stepCmd := _stepCmd + 1;
         END_IF 
       END_IF
     

  01:  // Wait for responce received
       IF ( _responseReceived )
       THEN
         // reset response received flag
        _responseReceived := FALSE;

         CASE  _response.State 
         OF
           CmdMessageState.BUFFERED : CommandBuffered := TRUE;
           CmdMessageState.DONE     : Done            := TRUE;
           CmdMessageState.ERROR    : Error           := TRUE;
         END_CASE
                
         // Done, Aborted or Error ?
         IF (_response.State >= CmdMessageState.DONE )
         THEN
           // Reset Busy flag
           Busy := FALSE;
           // Update results
           //OutCmd.Dummy := _response.Dummy;
           
           // set timeout
           SetTimeout(PT := _timeoutCmd, rTimer := _timerCmd);
           // inc step counter
          _stepCmd := _stepCmd + 1; 
         END_IF
       END_IF


  02: IF ( NOT Execute)
      THEN
        Reset();  
      END_IF     
      
ELSE
  // invalid step
  ErrorID := RobotLibraryEvents.ERR_INVALID_STEP;
END_CASE


// Reset FB
IF ( NOT Execute )
THEN
  Reset();
END_IF
END_METHOD

METHOD INTERNAL ParseResponsePayload : DINT
VAR_INPUT
  /// Response data
  ResponseData : RobotLibraryRecvDataFB;
  /// Timestamp
  Timestamp    : SystemTime;  
END_VAR
// Table 6-459: Received CMD payload (RC to PLC) of "ConfigureConveyor"
// --------------------------
// Header
// --------------------------
// Byte 00 : USINT      - ParSeq | State     
// Byte 01 : SINT       - AlarmMessageSeverity    
// Byte 02 : UINT       - AlarmMessageCode HB
// Byte 03 :            - AlarmMessageCode LB
// --------------------------
// call base implementation to parse the header from payload buffer
ResponseData.PayloadPtr := SUPER^.ParseResponsePayload(ResponseData := ResponseData, Timestamp := Timestamp);

// copy parsed header to response
_response.ParSeq                := _rspHeader.ParSeq;
_response.State                 := _rspHeader.State;
_response.AlarmMessageSeverity  := _rspHeader.AlarmMessageSeverity;
_response.AlarmMessageCode      := _rspHeader.AlarmMessageCode;

// Create logging
ParseResponsePayloadLog(ResponseData := ResponseData, Timestamp := Timestamp);
END_METHOD

METHOD INTERNAL ParseResponsePayloadLog
VAR_INPUT
  /// Response data
  ResponseData : RobotLibraryRecvDataFB;
  /// Timestamp
  Timestamp    : SystemTime;  
END_VAR
// Create log entry for Parameter start
CreateLogMessage      ( Timestamp   := Timestamp,
                        MessageType := MessageType.CMD,
                        Severity    := Severity.DEBUG,
                        MessageCode := 0,
                        MessageText := 'Parsed the following parameter(s) from response data:');
                        
// Create log entry for no parameter 
CreateLogMessage      ( Timestamp   := Timestamp,
                        MessageType := MessageType.CMD,
                        Severity    := Severity.DEBUG,
                        MessageCode := 0,
                        MessageText := 'This command has no parameter to parse...');
END_METHOD

METHOD PROTECTED Reset : DINT
VAR_INPUT
END_VAR
Reset := SUPER^.Reset();

Done               := FALSE;
Busy               := FALSE;
CommandBuffered    := FALSE;
END_METHOD

END_FUNCTION_BLOCK

// Library/POUs/ConveyorTracking/MC_RedefineTrackingPos/MC_RedefineTrackingPosFB
/// Redefine tracking position for conveyor tracking
FUNCTION_BLOCK MC_RedefineTrackingPosFB EXTENDS RobotLibraryBaseExecuteFB
// ------------------------------------------------------------------------- 
//  SRCI Robot Library                                                
// ------------------------------------------------------------------------- 
//                                                                           
//  Object:      RedefineTrackingPosFB                                       
//  Author:      Thorsten Brach                                                
//  Date:        2024-06-11
//
//  Description:                                              
//   
//                                                                           
//  Copyright: 
//    (C) 2024 Thorsten Brach. All rights reserved                                                                                                                                            
//             Licensed under the LGPL-3.0 license.
//                                                                           
//  Disclaimer:                                                                           
//    This project is provided without any guarantee and can be used for   
//    private and commercial purposes. Any use is at the user’s 
//    own risk and responsibility.
//
// -------------------------------------------------------------------------
VAR_INPUT
  /// Command parameter 
  ParCmd            : RedefineTrackingPosParCmd;      
END_VAR

VAR_OUTPUT
  /// Command is transferred and confirmed by the RC
  CommandBuffered   : BOOL;
  /// Receiving of input parameter values has been acknowledged by RC
  ParameterAccepted : BOOL;
  /// Command output 
  OutCmd            : RedefineTrackingPosOutCmd;    
END_VAR

VAR
  /// internal copy of command parameter 
 _parCmd            : RedefineTrackingPosParCmd;
  /// command data to send
 _command           : RedefineTrackingPosSendData;
  /// response data received
 _response          : RedefineTrackingPosRecvData;      
END_VAR

SUPER^(AxesGroup := AxesGroup);

METHOD PROTECTED CheckFunctionSupported : BOOL
VAR_IN_OUT
  /// Robot assignment of function
  AxesGroup : AxesGroup; 
END_VAR
CheckFunctionSupported := AxesGroup.InternalData.RCSupportedFunctions.RedefineTrackingPosition;

IF ( NOT CheckFunctionSupported )
THEN
  // call base implementation for set error and create log entry
  SUPER^.CheckFunctionSupported(AxesGroup := AxesGroup);
END_IF
END_METHOD

METHOD PROTECTED CheckParameterChanged : BOOL
VAR_IN_OUT
  /// Robot assignment of function
  AxesGroup : AxesGroup; 
END_VAR
// Check ParCmd Size is > 0, because MemCmp does not work correctly with size = 0
IF (SIZEOF(ParCmd) = 0) 
THEN 
  RETURN;
END_IF

// compare memory 
_parameterChanged := ( SysDepMemCmp(pData1 := ADR(ParCmd), pData2 := ADR(_parCmd), DataLen := SIZEOF(ParCmd)) <> RobotLibraryConstants.OK );

// check parameter valid ?
_parameterValid   := CheckParameterValid( AxesGroup := AxesGroup );

IF ((  _parameterChanged        )  AND 
    (  _parameterValid          )) OR
    (  _parameterUpdateInternal )  
THEN  
  // reset internal flag for send parameter update
 _parameterUpdateInternal := FALSE;
  // update internal copy of parameters 
 _parCmd := ParCmd;
  // inc parameter sequence
 _command.ParSeq := _command.ParSeq + 1;
  // update command data  
  CommandData := CreateCommandPayload(AxesGroup := AxesGroup); // ( Access via reference to rCommandFB in ACR )
  // notify active command register 
  AxesGroup.Acyclic.ActiveCommandRegister.NotifyParameterChanged := _uniqueID;
  // Reset parameter accepted flag
  ParameterAccepted := FALSE;  
END_IF
END_METHOD

METHOD INTERNAL CreateCommandPayload : RobotLibrarySendDataFB
VAR_IN_OUT
  /// Robot assignment of function
  AxesGroup : AxesGroup; 
END_VAR
// Table 6-444: Sent CMD payload (PLC to RC) of "RedefineTrackingPos"
// --------------------------
// Header
// --------------------------
// Byte 00 : UINT       - Type HB     
// Byte 01 :            - Type LB    
// Byte 02 : USINT      - Reserve | ExecutionMode
// Byte 03 : USINT      - ParSeq  | Priority
// --------------------------
// Datablock
// --------------------------
// Byte 04 : SINT       - EmitterID[0]
// Byte 05 : SINT       - EmitterID[1]
// Byte 06 : SINT       - EmitterID[2]
// Byte 07 : SINT       - EmitterID[3]
// Byte 08 : SINT       - ListenerID
// Byte 09 : BYTE       - Reserved
// Byte 10 : USINT      - ConveyorNo
// Byte 11 : USINT      - StartIndexInitPosition
// Byte 12 : REAL       - TrackingOffset HW HB
// Byte 13 :            - TrackingOffset HW LB
// Byte 14 :            - TrackingOffset LW HB
// Byte 15 :            - TrackingOffset LW LB
// Byte 16 : USINT      - FrameNo
// Byte 17 : USINT      - IndexTrackingOffset
// --------------------------
// set command parameter 
_command.CmdTyp                 :=  CmdType.RedefineTrackingPos;
_command.ExecMode               :=  ExecMode;
_command.ParSeq                 := _command.ParSeq;
_command.Priority               :=  Priority;
_command.EmitterID[0]           := 0; {warning 'ToDo'}
_command.EmitterID[1]           := 0; {warning 'ToDo'}
_command.EmitterID[2]           := 0; {warning 'ToDo'}
_command.EmitterID[3]           := 0; {warning 'ToDo'}
_command.ListenerID             := _parCmd.ListenerID;
_command.Reserve                := 0;
_command.ConveyorNo             := _parCmd.ConveyorNo;
_command.StartIndexInitPosition := _parCmd.StartIndexInitPosition;
_command.TrackingOffset         := _parCmd.TrackingOffset;
_command.FrameNo                := _parCmd.FrameNo;
_command.IndexTrackingOffset    := _parCmd.IndexTrackingOffset;

// copy command data to header
_cmdHeader := _command;
// call base implementation to copy header to payload buffer
CreateCommandPayload := SUPER^.CreateCommandPayload(AxesGroup := AxesGroup);


// add command.EmitterID[0]
CreateCommandPayload.AddSint(_command.EmitterID[0]);
// add command.EmitterID[1]
CreateCommandPayload.AddSint(_command.EmitterID[1]);
// add command.EmitterID[2]
CreateCommandPayload.AddSint(_command.EmitterID[2]);
// add command.EmitterID[3]
CreateCommandPayload.AddSint(_command.EmitterID[3]);
// add command.ListenerID
CreateCommandPayload.AddSint(_command.ListenerID);
// add command.Reserve
CreateCommandPayload.AddByte(_command.Reserve);
// add command.ConveyorNo
CreateCommandPayload.AddUsint(_command.ConveyorNo);
// add command.StartIndexInitPosition
CreateCommandPayload.AddUsint(_command.StartIndexInitPosition);
// add command.TrackingOffset
CreateCommandPayload.AddReal(_command.TrackingOffset);
// add command.FrameNo
CreateCommandPayload.AddUsint(_command.FrameNo);
// add command.IndexTrackingOffset
CreateCommandPayload.AddUsint(_command.IndexTrackingOffset);

// Create logging
CreateCommandPayloadLog(AxesGroup := AxesGroup);
END_METHOD

METHOD INTERNAL CreateCommandPayloadLog 
VAR_IN_OUT
  /// Robot assignment of function
  AxesGroup : AxesGroup; 
END_VAR
VAR 
  /// internal index for loops
 _idx : DINT;
END_VAR
// Create log entry for Parameter start
CreateLogMessage      ( Timestamp   := AxesGroup.InternalData.SystemTime,
                        MessageType := MessageType.CMD,
                        Severity    := Severity.DEBUG,
                        MessageCode := 0,
                        MessageText := 'Create command payload with the following parameter(s) :');

// Create log entry for EmitterID[x]
FOR _idx := 0 TO 3
DO
  CreateLogMessagePara2 ( Timestamp   := AxesGroup.InternalData.SystemTime,
                          MessageType := MessageType.CMD,
                          Severity    := Severity.DEBUG,
                          MessageCode := 0,
                          MessageText := 'Command.EmitterID[{2}] = {1}',
                          Para1       :=  SINT_TO_STRING(_command.EmitterID[_idx]),
                          Para2       :=  DINT_TO_STRING(_idx));
END_FOR

// Create log entry for ListenerID
CreateLogMessagePara1 ( Timestamp   := AxesGroup.InternalData.SystemTime,
                        MessageType := MessageType.CMD,
                        Severity    := Severity.DEBUG,
                        MessageCode := 0,
                        MessageText := 'Command.ListenerID = {1}',
                        Para1       :=  SINT_TO_STRING(_command.ListenerID));
                        
// Create log entry for Reserve
CreateLogMessagePara1 ( Timestamp   := AxesGroup.InternalData.SystemTime,
                        MessageType := MessageType.CMD,
                        Severity    := Severity.DEBUG,
                        MessageCode := 0,
                        MessageText := 'Command.Reserve = {1}',
                        Para1       :=  BYTE_TO_STRING(_command.Reserve));

// Create log entry for ConveyorNo
CreateLogMessagePara1 ( Timestamp   := AxesGroup.InternalData.SystemTime,
                        MessageType := MessageType.CMD,
                        Severity    := Severity.DEBUG,
                        MessageCode := 0,
                        MessageText := 'Command.ConveyorNo = {1}',
                        Para1       :=  USINT_TO_STRING(_command.ConveyorNo));

// Create log entry for StartIndexInitPosition
CreateLogMessagePara1 ( Timestamp   := AxesGroup.InternalData.SystemTime,
                        MessageType := MessageType.CMD,
                        Severity    := Severity.DEBUG,
                        MessageCode := 0,
                        MessageText := 'Command.StartIndexInitPosition = {1}',
                        Para1       :=  USINT_TO_STRING(_command.StartIndexInitPosition));

// Create log entry for TrackingOffset
CreateLogMessagePara1 ( Timestamp   := AxesGroup.InternalData.SystemTime,
                        MessageType := MessageType.CMD,
                        Severity    := Severity.DEBUG,
                        MessageCode := 0,
                        MessageText := 'Command.TrackingOffset = {1}',
                        Para1       :=  REAL_TO_STRING(_command.TrackingOffset));

// Create log entry for FrameNo
CreateLogMessagePara1 ( Timestamp   := AxesGroup.InternalData.SystemTime,
                        MessageType := MessageType.CMD,
                        Severity    := Severity.DEBUG,
                        MessageCode := 0,
                        MessageText := 'Command.FrameNo = {1}',
                        Para1       :=  USINT_TO_STRING(_command.FrameNo));

// Create log entry for IndexTrackingOffset
CreateLogMessagePara1 ( Timestamp   := AxesGroup.InternalData.SystemTime,
                        MessageType := MessageType.CMD,
                        Severity    := Severity.DEBUG,
                        MessageCode := 0,
                        MessageText := 'Command.IndexTrackingOffset = {1}',
                        Para1       :=  USINT_TO_STRING(_command.IndexTrackingOffset));
END_METHOD

METHOD FB_init : BOOL
VAR_INPUT
  /// if TRUE, the retain variables are initialized (warm start / cold start)
  bInitRetains : BOOL; 
  /// if TRUE, the instance afterwards gets moved into the copy code (online change)
  bInCopyCode  : BOOL;  
END_VAR
MyType := 'MC_RedefineTrackingPosFB';
END_METHOD

METHOD PROTECTED OnCall
VAR_IN_OUT
  /// Robot assignment of function
  AxesGroup : AxesGroup; 
END_VAR
// call base implementation
SUPER^.OnCall(AxesGroup := AxesGroup);

CASE _stepCmd OF
  
  00:  IF ( _execute_R.Q )  
       THEN
         // Check function is supported and parameter are valid ?
         IF (( CheckFunctionSupported( AxesGroup := AxesGroup )) AND
             ( CheckParameterValid   ( AxesGroup := AxesGroup )))      
         THEN
           // set busy flag
           Busy := TRUE;
           // Reset command outputs
           SysDepMemSet(pDest := ADR(OutCmd), Value := 0, DataLen := SIZEOF(OutCmd));         
           // apply command parameter
          _parCmd := ParCmd;
           // init parameter sequence
          _command.ParSeq := 1;
           // create command data
           CommandData := CreateCommandPayload(AxesGroup := AxesGroup);
           // Add command to active command register
          _uniqueID := AxesGroup.Acyclic.ActiveCommandRegister.AddCmd( pCommandFB := ADR(THIS^ ));     
           // set timeout
           SetTimeout(PT := _timeoutCmd, rTimer := _timerCmd);
           // inc step counter
          _stepCmd := _stepCmd + 1; 
         END_IF
       END_IF
     

  01:  // Wait for responce received
       IF ( _responseReceived )
       THEN
         // reset response received flag
        _responseReceived := FALSE;

         CASE  _response.State 
         OF
           CmdMessageState.BUFFERED : CommandBuffered   := TRUE;
           CmdMessageState.ACTIVE   : ParameterAccepted := TRUE;
           CmdMessageState.DONE     : Done              := TRUE;
           CmdMessageState.ERROR    : Error             := TRUE;
         END_CASE
                
         // Done, Aborted or Error ?
         IF (_response.State >= CmdMessageState.DONE )
         THEN
           // Reset Busy flag
           Busy := FALSE;
           // Update results
           OutCmd.OriginID          := _response.OriginID;
           OutCmd.InvocationCounter := _response.InvocationCounter;
           // set timeout
           SetTimeout(PT := _timeoutCmd, rTimer := _timerCmd);
           // inc step counter
          _stepCmd := _stepCmd + 1; 
         END_IF
       END_IF


  02: IF ( NOT Execute)
      THEN
        Reset();
      END_IF
     
ELSE
  // invalid step
  ErrorID := RobotLibraryEvents.ERR_INVALID_STEP;
END_CASE


// Reset FB
IF ( NOT Execute )
THEN
  Reset();
END_IF
END_METHOD

METHOD INTERNAL ParseResponsePayload : DINT
VAR_INPUT
  /// Response data
  ResponseData : RobotLibraryRecvDataFB;
  /// Timestamp
  Timestamp    : SystemTime;  
END_VAR
// Table 6-445: Received CMD payload (RC to PLC) of "RedefineTrackingPos"
// --------------------------
// Header
// --------------------------
// Byte 00 : USINT      - ParSeq | State     
// Byte 01 : SINT       - AlarmMessageSeverity    
// Byte 02 : UINT       - AlarmMessageCode HB
// Byte 03 :            - AlarmMessageCode LB
// --------------------------
// Datablock
// --------------------------
// Byte 04 : USINT InvocationCounter;
// Byte 05 : SINT  Reserved;
// Byte 06 : INT   OriginID;
// Byte 07 :       OriginID;
// call base implementation to parse the header from payload buffer
ResponseData.PayloadPtr := SUPER^.ParseResponsePayload(ResponseData := ResponseData, Timestamp := Timestamp);

// copy parsed header to response
_response.ParSeq                := _rspHeader.ParSeq;
_response.State                 := _rspHeader.State;
_response.AlarmMessageSeverity  := _rspHeader.AlarmMessageSeverity;
_response.AlarmMessageCode      := _rspHeader.AlarmMessageCode;

// Get Response.InvocationCounter
_response.InvocationCounter := ResponseData.GetUsint();
// Get Response.Reserved
_response.Reserved := ResponseData.GetSint();
// Get Response.InvocationCounter
_response.OriginID := ResponseData.GetInt();

// Create logging
ParseResponsePayloadLog(ResponseData := ResponseData, Timestamp := Timestamp);
END_METHOD

METHOD INTERNAL ParseResponsePayloadLog
VAR_INPUT
  /// Response data
  ResponseData : RobotLibraryRecvDataFB;
  /// Timestamp
  Timestamp    : SystemTime;  
END_VAR
// Create log entry for Parameter start
CreateLogMessage      ( Timestamp   := Timestamp,
                        MessageType := MessageType.CMD,
                        Severity    := Severity.DEBUG,
                        MessageCode := 0,
                        MessageText := 'Parsed the following parameter(s) from response data:');
                        
// Create log entry for InvocationCounter
CreateLogMessagePara1 ( Timestamp   := Timestamp,
                        MessageType := MessageType.CMD,
                        Severity    := Severity.DEBUG,
                        MessageCode := 0,
                        MessageText := 'Response.InvocationCounter = {1}',
                        Para1       :=  USINT_TO_STRING(_response.InvocationCounter));

// Create log entry for Reserve
CreateLogMessagePara1 ( Timestamp   := Timestamp,
                        MessageType := MessageType.CMD,
                        Severity    := Severity.DEBUG,
                        MessageCode := 0,
                        MessageText := 'Response.Reserve = {1}',
                        Para1       :=  SINT_TO_STRING(_response.Reserved));

// Create log entry for OriginID
CreateLogMessagePara1 ( Timestamp   := Timestamp,
                        MessageType := MessageType.CMD,
                        Severity    := Severity.DEBUG,
                        MessageCode := 0,
                        MessageText := 'Response.OriginID = {1}',
                        Para1       :=  INT_TO_STRING(_response.OriginID));
END_METHOD

METHOD PROTECTED Reset : DINT
VAR_INPUT
END_VAR
Reset := SUPER^.Reset();

Done               := FALSE;
Busy               := FALSE;
CommandBuffered    := FALSE;
ParameterAccepted  := FALSE;
END_METHOD

END_FUNCTION_BLOCK

// Library/POUs/ConveyorTracking/MC_SyncToConveyor/MC_SyncToConveyorFB
/// Synchronize robot with conveyor
FUNCTION_BLOCK MC_SyncToConveyorFB EXTENDS RobotLibraryBaseEnableFB
// ------------------------------------------------------------------------- 
//  SRCI Robot Library                                                
// ------------------------------------------------------------------------- 
//                                                                           
//  Object:      SyncToConveyorFB                                       
//  Author:      Thorsten Brach                                                
//  Date:        2024-06-11
//
//  Description:                                              
//   
//                                                                           
//  Copyright: 
//    (C) 2024 Thorsten Brach. All rights reserved                                                                                                                                            
//             Licensed under the LGPL-3.0 license.
//                                                                           
//  Disclaimer:                                                                           
//    This project is provided without any guarantee and can be used for   
//    private and commercial purposes. Any use is at the user’s 
//    own risk and responsibility.
//
// -------------------------------------------------------------------------
VAR_INPUT
  /// Command parameter 
  ParCmd            : SyncToConveyorParCmd;      
END_VAR

VAR_OUTPUT
  /// Command is transferred and confirmed by the RC
  CommandBuffered   : BOOL;
  /// The command takes control of the motion of the according axis group
  Active            : BOOL;
  /// The command was aborted by another command.
  CommandAborted    : BOOL;
  /// Receiving of input parameter values has been acknowledged by RC
  ParameterAccepted : BOOL;
  /// Command output 
  OutCmd            : SyncToConveyorOutCmd;      
END_VAR

VAR
  /// internal copy of command parameter 
 _parCmd            : SyncToConveyorParCmd;
  /// command data to send
 _command           : SyncToConveyorSendData;
  /// response data received
 _response          : SyncToConveyorRecvData;      
END_VAR

SUPER^(AxesGroup := AxesGroup);

METHOD PROTECTED CheckFunctionSupported : BOOL
VAR_IN_OUT
  /// Robot assignment of function
  AxesGroup : AxesGroup; 
END_VAR
CheckFunctionSupported := AxesGroup.InternalData.RCSupportedFunctions.SyncToConveyor;

IF ( NOT CheckFunctionSupported )
THEN
  // call base implementation for set error and create log entry
  SUPER^.CheckFunctionSupported(AxesGroup := AxesGroup);
END_IF
END_METHOD

METHOD PROTECTED CheckParameterChanged : BOOL
VAR_IN_OUT
  /// Robot assignment of function
  AxesGroup    : AxesGroup; 
END_VAR
// Check ParCmd Size is > 0, because MemCmp does not work correctly with size = 0
IF (SIZEOF(ParCmd) = 0) 
THEN 
  RETURN;
END_IF

// compare memory 
_parameterChanged := ( SysDepMemCmp(pData1 := ADR(ParCmd), pData2 := ADR(_parCmd), DataLen := SIZEOF(ParCmd)) <> RobotLibraryConstants.OK );

// check parameter valid ?
_parameterValid   := CheckParameterValid( AxesGroup := AxesGroup );

IF ((  _parameterChanged        )  AND 
    (  _parameterValid          )) OR
    (  _parameterUpdateInternal )  
THEN  
  // reset internal flag for send parameter update
 _parameterUpdateInternal := FALSE;
  // update internal copy of parameters 
 _parCmd := ParCmd;
  // inc parameter sequence
 _command.ParSeq := _command.ParSeq + 1;
  // update command data  
  CommandData := CreateCommandPayload(AxesGroup := AxesGroup); // ( Access via reference to rCommandFB in ACR )
  // notify active command register 
  AxesGroup.Acyclic.ActiveCommandRegister.NotifyParameterChanged := _uniqueID;
  // Reset parameter accepted flag
  ParameterAccepted := FALSE;  
END_IF
END_METHOD

METHOD INTERNAL CreateCommandPayload : RobotLibrarySendDataFB
VAR_IN_OUT
  /// Robot assignment of function
  AxesGroup : AxesGroup; 
END_VAR
// Table 6-452: Sent CMD payload (PLC to RC) of "SyncToConveyor"
// --------------------------
// Header
// --------------------------
// Byte 00 : UINT       - Type HB     
// Byte 01 :            - Type LB    
// Byte 02 : USINT      - Reserve | ExecutionMode
// Byte 03 : USINT      - ParSeq  | Priority
// --------------------------
// Datablock
// --------------------------
// Byte 04 : SINT       - EmitterID[0]
// Byte 05 : SINT       - EmitterID[1]
// Byte 06 : SINT       - EmitterID[2]
// Byte 07 : SINT       - EmitterID[3]
// Byte 08 : SINT       - ListenerID
// Byte 09 : BYTE       - Reserved
// Byte 10 : USINT      - ConveyorNo
// Byte 11 : USINT      - FrameNo
// Byte 12 : USINT      - SyncInMode
// Byte 13 : REAL       - SyncInParameter HW HB
// Byte 14 :            - SyncInParameter HW LB
// Byte 15 :            - SyncInParameter LW HB
// Byte 16 :            - SyncInParameter LW LB
// Byte 17 : REAL       - MaxVelocity     HW HB
// Byte 18 :            - MaxVelocity     HW LB
// Byte 19 :            - MaxVelocity     LW HB
// Byte 20 :            - MaxVelocity     LW LB
// Byte 21 : REAL       - MaxAcceleration HW HB
// Byte 22 :            - MaxAcceleration HW LB
// Byte 23 :            - MaxAcceleration LW HB
// Byte 24 :            - MaxAcceleration LW LB
// --------------------------
// set command parameter 
_command.CmdTyp          :=  CmdType.SyncToConveyor;
_command.ExecMode        :=  ExecMode;
_command.ParSeq          := _command.ParSeq;
_command.Priority        :=  Priority;
_command.EmitterID[0]    := 0; {warning 'ToDo'}
_command.EmitterID[1]    := 0; {warning 'ToDo'}
_command.EmitterID[2]    := 0; {warning 'ToDo'}
_command.EmitterID[3]    := 0; {warning 'ToDo'}
_command.ListenerID      := _parCmd.ListenerID;
_command.Reserve         := 0;
_command.ConveyorNo      := _parCmd.ConveyorNo;
_command.FrameNo         := _parCmd.FrameNo;
_command.SyncInMode      := _parCmd.SyncInMode;
_command.SyncInParameter := _parCmd.SyncInParameter;
_command.MaxVelocity     := _parCmd.MaxVelocity;
_command.MaxAcceleration := _parCmd.MaxAcceleration;

// copy command data to header
_cmdHeader := _command;
// call base implementation to copy header to payload buffer
CreateCommandPayload := SUPER^.CreateCommandPayload(AxesGroup := AxesGroup);


// add command.EmitterID[0]
CreateCommandPayload.AddSint(_command.EmitterID[0]);
// add command.EmitterID[1]
CreateCommandPayload.AddSint(_command.EmitterID[1]);
// add command.EmitterID[2]
CreateCommandPayload.AddSint(_command.EmitterID[2]);
// add command.EmitterID[3]
CreateCommandPayload.AddSint(_command.EmitterID[3]);
// add command.ListenerID
CreateCommandPayload.AddSint(_command.ListenerID);
// add command.Reserve
CreateCommandPayload.AddByte(_command.Reserve);
// add command.ConveyorNo
CreateCommandPayload.AddUsint(_command.ConveyorNo);
// add command.FrameNo
CreateCommandPayload.AddUsint(_command.FrameNo);
// add command.SyncInMode
CreateCommandPayload.AddUsint(_command.SyncInMode);
// add command.SyncInParameter
CreateCommandPayload.AddReal(_command.SyncInParameter);
// add command.MaxVelocity
CreateCommandPayload.AddReal(_command.MaxVelocity);
// add command.MaxAcceleration
CreateCommandPayload.AddReal(_command.MaxAcceleration);

// Create logging
CreateCommandPayloadLog(AxesGroup := AxesGroup);
END_METHOD

METHOD INTERNAL CreateCommandPayloadLog 
VAR_IN_OUT
  /// Robot assignment of function
  AxesGroup : AxesGroup; 
END_VAR
VAR 
  /// internal index for loops
 _idx : DINT;
END_VAR
// Create log entry for Parameter start
CreateLogMessage      ( Timestamp   := AxesGroup.InternalData.SystemTime,
                        MessageType := MessageType.CMD,
                        Severity    := Severity.DEBUG,
                        MessageCode := 0,
                        MessageText := 'Create command payload with the following parameter(s) :');

// Create log entry for EmitterID[x]
FOR _idx := 0 TO 3
DO
  CreateLogMessagePara2 ( Timestamp   := AxesGroup.InternalData.SystemTime,
                          MessageType := MessageType.CMD,
                          Severity    := Severity.DEBUG,
                          MessageCode := 0,
                          MessageText := 'Command.EmitterID[{2}] = {1}',
                          Para1       :=  SINT_TO_STRING(_command.EmitterID[_idx]),
                          Para2       :=  DINT_TO_STRING(_idx));
END_FOR

// Create log entry for ListenerID
CreateLogMessagePara1 ( Timestamp   := AxesGroup.InternalData.SystemTime,
                        MessageType := MessageType.CMD,
                        Severity    := Severity.DEBUG,
                        MessageCode := 0,
                        MessageText := 'Command.ListenerID = {1}',
                        Para1       :=  SINT_TO_STRING(_command.ListenerID));
                        
// Create log entry for Reserve
CreateLogMessagePara1 ( Timestamp   := AxesGroup.InternalData.SystemTime,
                        MessageType := MessageType.CMD,
                        Severity    := Severity.DEBUG,
                        MessageCode := 0,
                        MessageText := 'Command.Reserve = {1}',
                        Para1       :=  BYTE_TO_STRING(_command.Reserve));

// Create log entry for ConveyorNo
CreateLogMessagePara1 ( Timestamp   := AxesGroup.InternalData.SystemTime,
                        MessageType := MessageType.CMD,
                        Severity    := Severity.DEBUG,
                        MessageCode := 0,
                        MessageText := 'Command.ConveyorNo = {1}',
                        Para1       :=  USINT_TO_STRING(_command.ConveyorNo));
                        
// Create log entry for FrameNo
CreateLogMessagePara1 ( Timestamp   := AxesGroup.InternalData.SystemTime,
                        MessageType := MessageType.CMD,
                        Severity    := Severity.DEBUG,
                        MessageCode := 0,
                        MessageText := 'Command.FrameNo = {1}',
                        Para1       :=  USINT_TO_STRING(_command.FrameNo));       
                        
// Create log entry for SyncInMode
CreateLogMessagePara1 ( Timestamp   := AxesGroup.InternalData.SystemTime,
                        MessageType := MessageType.CMD,
                        Severity    := Severity.DEBUG,
                        MessageCode := 0,
                        MessageText := 'Command.SyncInMode = {1}',
                        Para1       :=  SYNC_IN_MODE_TO_STRING(_command.SyncInMode));                                         
                        
// Create log entry for SyncInParameter
CreateLogMessagePara1 ( Timestamp   := AxesGroup.InternalData.SystemTime,
                        MessageType := MessageType.CMD,
                        Severity    := Severity.DEBUG,
                        MessageCode := 0,
                        MessageText := 'Command.SyncInParameter = {1}',
                        Para1       :=  REAL_TO_STRING(_command.SyncInParameter));                                                                 

// Create log entry for MaxVelocity
CreateLogMessagePara1 ( Timestamp   := AxesGroup.InternalData.SystemTime,
                        MessageType := MessageType.CMD,
                        Severity    := Severity.DEBUG,
                        MessageCode := 0,
                        MessageText := 'Command.MaxVelocity = {1}',
                        Para1       :=  REAL_TO_STRING(_command.MaxVelocity));                                                                 

// Create log entry for MaxAcceleration
CreateLogMessagePara1 ( Timestamp   := AxesGroup.InternalData.SystemTime,
                        MessageType := MessageType.CMD,
                        Severity    := Severity.DEBUG,
                        MessageCode := 0,
                        MessageText := 'Command.MaxAcceleration = {1}',
                        Para1       :=  REAL_TO_STRING(_command.MaxAcceleration));
END_METHOD

METHOD FB_init : BOOL
VAR_INPUT
  /// if TRUE, the retain variables are initialized (warm start / cold start)
  bInitRetains : BOOL; 
  /// if TRUE, the instance afterwards gets moved into the copy code (online change)
  bInCopyCode  : BOOL;  
END_VAR
MyType := 'MC_SyncToConveyorFB';
END_METHOD

METHOD PROTECTED OnCall
VAR_IN_OUT
  /// Robot assignment of function
  AxesGroup : AxesGroup; 
END_VAR
// call base implementation
SUPER^.OnCall(AxesGroup := AxesGroup);

CASE _stepCmd OF
  
  00:  IF ( _enable_R.Q ) 
       THEN
         // reset the rising edge
        _enable_R();       
         // reset the falling edge
        _enable_F();     

         // Check function is supported and parameter are valid ?
         IF (( CheckFunctionSupported( AxesGroup := AxesGroup )) AND
             ( CheckParameterValid   ( AxesGroup := AxesGroup )))      
         THEN
           // set busy flag
           Busy := TRUE;
           // Reset command outputs
           SysDepMemSet(pDest := ADR(OutCmd), Value := 0, DataLen := SIZEOF(OutCmd));         
           // apply command parameter
          _parCmd := ParCmd;
           // init parameter sequence
          _command.ParSeq := 1;
           // create command data
           CommandData := CreateCommandPayload(AxesGroup := AxesGroup);
           // Add command to active command register
          _uniqueID := AxesGroup.Acyclic.ActiveCommandRegister.AddCmd( pCommandFB := ADR(THIS^ ));     
           // set timeout
           SetTimeout(PT := _timeoutCmd, rTimer := _timerCmd);
           // inc step counter
          _stepCmd := _stepCmd + 1;
         END_IF 
       END_IF
     

  01:  // Wait for responce received
       IF ( _responseReceived )
       THEN
         // reset response received flag
        _responseReceived := FALSE;

         CASE  _response.State 
         OF
           CmdMessageState.BUFFERED    : CommandBuffered    := TRUE;
           CmdMessageState.ACTIVE      : ParameterAccepted  := TRUE;
                                         Active             := TRUE; {warning 'ToDo'}           
           CmdMessageState.ABORTED     : CommandAborted     := TRUE;
           CmdMessageState.ERROR       : Error              := TRUE;
         END_CASE
                
         // Update results
         OutCmd.InvocationCounter := _response.InvocationCounter;
         OutCmd.OriginID          := _response.OriginID;
         OutCmd.InSync            := _response.InSync;           
         Enabled                  := TRUE; {warning 'ToDo'}
                
         // Done, Aborted or Error ?
         IF (_response.State >= CmdMessageState.DONE )
         THEN
           // reset busy flag
           Enabled := FALSE; 
           // set timeout
           SetTimeout(PT := _timeoutCmd, rTimer := _timerCmd);
           // inc step counter
          _stepCmd := _stepCmd + 1; 
         END_IF
       END_IF

       // do not abort directly, so that the ParSeq update can be send
       IF ( _enable_R.Q ) OR ( _enable_F.Q ) 
       THEN
         // trigger parameter update to disable FB
        _parameterUpdateInternal := TRUE;
         // reset the rising edge
        _enable_R();       
         // reset the falling edge
        _enable_F();       
       END_IF


  02:  IF (NOT Enable)
       THEN
         Reset();  
       END_IF


ELSE
  // invalid step
  ErrorID := RobotLibraryEvents.ERR_INVALID_STEP;
END_CASE



// Reset FB
IF (( _enable_R.Q ) OR
    ( _enable_F.Q ))
THEN
  Reset(); 
END_IF
END_METHOD

METHOD INTERNAL ParseResponsePayload : DINT
VAR_INPUT
  /// Response data
  ResponseData : RobotLibraryRecvDataFB;
  /// Timestamp
  Timestamp    : SystemTime;  
END_VAR
// Table 6-453: Received CMD payload (RC to PLC) of "SyncToConveyor"
// --------------------------
// Header
// --------------------------
// Byte 00 : USINT      - ParSeq | State     
// Byte 01 : SINT       - AlarmMessageSeverity    
// Byte 02 : UINT       - AlarmMessageCode HB
// Byte 03 :            - AlarmMessageCode LB
// --------------------------
// Datablock
// --------------------------
// Byte 04 : USINT       - InvocationCounter
// Byte 05 : SINT        - Reserved
// Byte 06 : INT         - OriginID
// Byte 07 : BOOL        - InSync
// --------------------------
// call base implementation to parse the header from payload buffer
ResponseData.PayloadPtr := SUPER^.ParseResponsePayload(ResponseData := ResponseData, Timestamp := Timestamp);

// copy parsed header to response
_response.ParSeq                := _rspHeader.ParSeq;
_response.State                 := _rspHeader.State;
_response.AlarmMessageSeverity  := _rspHeader.AlarmMessageSeverity;
_response.AlarmMessageCode      := _rspHeader.AlarmMessageCode;

// Get Response.InvocationCounter
_response.InvocationCounter := ResponseData.GetUsint();
// Get Response.Reserved
_response.Reserved := ResponseData.GetSint();
// Get Response.InvocationCounter
_response.OriginID := ResponseData.GetInt();
// Get Response.InSync
_response.InSync   := ResponseData.GetBool();

// Create logging
ParseResponsePayloadLog(ResponseData := ResponseData, Timestamp := Timestamp);
END_METHOD

METHOD INTERNAL ParseResponsePayloadLog
VAR_INPUT
  /// Response data
  ResponseData : RobotLibraryRecvDataFB;
  /// Timestamp
  Timestamp    : SystemTime;  
END_VAR
// Create log entry for Parameter start
CreateLogMessage      ( Timestamp   := Timestamp,
                        MessageType := MessageType.CMD,
                        Severity    := Severity.DEBUG,
                        MessageCode := 0,
                        MessageText := 'Parsed the following parameter(s) from response data:');
                        
// Create log entry for InvocationCounter
CreateLogMessagePara1 ( Timestamp   := Timestamp,
                        MessageType := MessageType.CMD,
                        Severity    := Severity.DEBUG,
                        MessageCode := 0,
                        MessageText := 'Response.InvocationCounter = {1}',
                        Para1       :=  USINT_TO_STRING(_response.InvocationCounter));

// Create log entry for Reserve
CreateLogMessagePara1 ( Timestamp   := Timestamp,
                        MessageType := MessageType.CMD,
                        Severity    := Severity.DEBUG,
                        MessageCode := 0,
                        MessageText := 'Response.Reserve = {1}',
                        Para1       :=  SINT_TO_STRING(_response.Reserved));

// Create log entry for OriginID
CreateLogMessagePara1 ( Timestamp   := Timestamp,
                        MessageType := MessageType.CMD,
                        Severity    := Severity.DEBUG,
                        MessageCode := 0,
                        MessageText := 'Response.OriginID = {1}',
                        Para1       :=  INT_TO_STRING(_response.OriginID));

// Create log entry for InSync
CreateLogMessagePara1 ( Timestamp   := Timestamp,
                        MessageType := MessageType.CMD,
                        Severity    := Severity.DEBUG,
                        MessageCode := 0,
                        MessageText := 'Response.InSync = {1}',
                        Para1       :=  BOOL_TO_STRING(_response.InSync));
END_METHOD

METHOD PROTECTED Reset : DINT
VAR_INPUT
END_VAR
SUPER^.Reset();

Busy               := FALSE;
Active             := FALSE;
CommandBuffered    := FALSE;
CommandAborted     := FALSE;
ParameterAccepted  := FALSE;
END_METHOD

END_FUNCTION_BLOCK

// Library/POUs/ForceControl/MC_ForceControl/MC_ForceControlFB
/// Enables the RC to apply user defined force/ torque through RA’s TCP movement
FUNCTION_BLOCK MC_ForceControlFB EXTENDS RobotLibraryBaseFB
// ------------------------------------------------------------------------- 
//  SRCI Robot Library                                                
// ------------------------------------------------------------------------- 
//                                                                           
//  Object:      ForceControlFB                                       
//  Author:      Thorsten Brach                                                
//  Date:        2024-06-01
//
//  Description:                                              
//   
//                                                                           
//  Copyright: 
//    (C) 2024 Thorsten Brach. All rights reserved                                                                                                                                            
//             Licensed under the LGPL-3.0 license.
//                                                                           
//  Disclaimer:                                                                           
//    This project is provided without any guarantee and can be used for   
//    private and commercial purposes. Any use is at the user’s 
//    own risk and responsibility.
//
// -------------------------------------------------------------------------
VAR_INPUT
  /// Set TRUE to activate ForceControl
  Enable             : BOOL;
  /// Command parameter 
  ParCmd             : ForceControlParCmd;      
END_VAR

VAR_OUTPUT
  /// TRUE, while the following outputs return valid values:
  /// - ForceStatus
  Valid              : BOOL;
  /// FB is being processed
  Busy               : BOOL;
  /// Command is transferred and confirmed by the RC
  CommandBuffered    : BOOL;
  /// Receiving of input parameter values has been acknowledged by RC
  ParameterAccepted  : BOOL;
  /// Command output 
  OutCmd             : ForceControlOutCmd;    
END_VAR

VAR
  /// internal copy of command parameter 
 _parCmd            : ForceControlParCmd;
  /// command data to send
 _command           : ForceControlSendData;
  /// response data received
 _response          : ForceControlRecvData;      
  /// Rising edge for enable
 _enable_R          : R_TRIG;
  /// Falling edge for enable
 _enable_F          : F_TRIG;  
END_VAR

SUPER^(AxesGroup := AxesGroup);

METHOD PROTECTED CheckFunctionSupported : BOOL
VAR_IN_OUT
  /// Robot assignment of function
  AxesGroup : AxesGroup; 
END_VAR
CheckFunctionSupported := AxesGroup.InternalData.RCSupportedFunctions.ForceControl;

IF ( NOT CheckFunctionSupported )
THEN
  // call base implementation for set error and create log entry
  SUPER^.CheckFunctionSupported(AxesGroup := AxesGroup);
END_IF
END_METHOD

METHOD PROTECTED CheckParameterChanged : BOOL
VAR_IN_OUT
  /// Robot assignment of function
  AxesGroup    : AxesGroup; 
END_VAR
// Check ParCmd Size is > 0, because MemCmp does not work correctly with size = 0
IF (SIZEOF(ParCmd) = 0) 
THEN 
  RETURN;
END_IF

// compare memory 
_parameterChanged := ( SysDepMemCmp(pData1 := ADR(ParCmd), pData2 := ADR(_parCmd), DataLen := SIZEOF(ParCmd)) <> RobotLibraryConstants.OK );

// check parameter valid ?
_parameterValid   := CheckParameterValid( AxesGroup := AxesGroup );

IF ((  _parameterChanged        )  AND 
    (  _parameterValid          )) OR
    (  _parameterUpdateInternal )  
THEN  
  // reset internal flag for send parameter update
 _parameterUpdateInternal := FALSE;
  // update internal copy of parameters 
 _parCmd := ParCmd;
  // inc parameter sequence
 _command.ParSeq := _command.ParSeq + 1;
  // update command data  
  CommandData := CreateCommandPayload(AxesGroup := AxesGroup); // ( Access via reference to rCommandFB in ACR )
  // notify active command register 
  AxesGroup.Acyclic.ActiveCommandRegister.NotifyParameterChanged := _uniqueID;
  // Reset parameter accepted flag
  ParameterAccepted := FALSE;  
END_IF
END_METHOD

METHOD INTERNAL CreateCommandPayload : RobotLibrarySendDataFB
VAR_IN_OUT
  /// Robot assignment of function
  AxesGroup : AxesGroup; 
END_VAR
// Table 6-719: Sent CMD payload (PLC to RC) of "ForceControl"
// --------------------------
// Header
// --------------------------
// Byte 00 : UINT       - Type HB     
// Byte 01 :            - Type LB    
// Byte 02 : USINT      - Reserve | ExecutionMode
// Byte 03 : USINT      - ParSeq  | Priority
// --------------------------
// Datablock
// --------------------------
// Byte 004 : USINT      - ToolNo 
// Byte 005 : USINT      - FrameNo 
// Byte 006 : USINT      - ConnectionMode 
// Byte 007 : BOOL       - FixedSensor
// Byte 008 : REAL       - SensorFrame[0] HW HB
// Byte 009 :            - SensorFrame[0] HW LB
// Byte 010 :            - SensorFrame[0] LW HB
// Byte 011 :            - SensorFrame[0] LW LB
// Byte 012 : REAL       - SensorFrame[1] HW HB
// Byte 013 :            - SensorFrame[1] HW LB
// Byte 014 :            - SensorFrame[1] LW HB
// Byte 015 :            - SensorFrame[1] LW LB
// Byte 016 : REAL       - SensorFrame[2] HW HB
// Byte 017 :            - SensorFrame[2] HW LB
// Byte 018 :            - SensorFrame[2] LW HB
// Byte 019 :            - SensorFrame[2] LW LB
// Byte 020 : REAL       - SensorFrame[3] HW HB
// Byte 021 :            - SensorFrame[3] HW LB
// Byte 022 :            - SensorFrame[3] LW HB
// Byte 023 :            - SensorFrame[3] LW LB
// Byte 024 : REAL       - SensorFrame[4] HW HB
// Byte 025 :            - SensorFrame[4] HW LB
// Byte 026 :            - SensorFrame[4] LW HB
// Byte 027 :            - SensorFrame[4] LW LB
// Byte 028 : REAL       - SensorFrame[5] HW HB
// Byte 029 :            - SensorFrame[5] HW LB
// Byte 030 :            - SensorFrame[5] LW HB
// Byte 031 :            - SensorFrame[5] LW LB
// Byte 032 :            - CalibrationData
// Byte 033 :            - ReferenceType
// Byte 034 : REAL       - SensorValue[0] HW HB
// Byte 035 :            - SensorValue[0] HW LB
// Byte 036 :            - SensorValue[0] LW HB
// Byte 037 :            - SensorValue[0] LW LB
// Byte 038 : REAL       - SensorValue[1] HW HB
// Byte 039 :            - SensorValue[1] HW LB
// Byte 040 :            - SensorValue[1] LW HB
// Byte 041 :            - SensorValue[1] LW LB
// Byte 042 : REAL       - SensorValue[2] HW HB
// Byte 043 :            - SensorValue[2] HW LB
// Byte 044 :            - SensorValue[2] LW HB
// Byte 045 :            - SensorValue[2] LW LB
// Byte 046 : REAL       - SensorValue[3] HW HB
// Byte 047 :            - SensorValue[3] HW LB
// Byte 048 :            - SensorValue[3] LW HB
// Byte 049 :            - SensorValue[3] LW LB
// Byte 050 : REAL       - SensorValue[4] HW HB
// Byte 051 :            - SensorValue[4] HW LB
// Byte 052 :            - SensorValue[4] LW HB
// Byte 053 :            - SensorValue[4] LW LB
// Byte 054 : REAL       - SensorValue[5] HW HB
// Byte 055 :            - SensorValue[5] HW LB
// Byte 056 :            - SensorValue[5] LW HB
// Byte 057 :            - SensorValue[5] LW LB
// Byte 058 : REAL       - SensorValue[5] HW HB
// Byte 059 :            - SensorValue[5] HW LB
// Byte 060 :            - SensorValue[5] LW HB
// Byte 061 :            - SensorValue[5] LW LB
// Byte 062 : REAL       - TargetValue[0] HW HB
// Byte 063 :            - TargetValue[0] HW LB
// Byte 064 :            - TargetValue[0] LW HB
// Byte 065 :            - TargetValue[0] LW LB
// Byte 066 : REAL       - TargetValue[1] HW HB
// Byte 067 :            - TargetValue[1] HW LB
// Byte 068 :            - TargetValue[1] LW HB
// Byte 069 :            - TargetValue[1] LW LB
// Byte 070 : REAL       - TargetValue[2] HW HB
// Byte 071 :            - TargetValue[2] HW LB
// Byte 072 :            - TargetValue[2] LW HB
// Byte 073 :            - TargetValue[2] LW LB
// Byte 074 : REAL       - TargetValue[3] HW HB
// Byte 075 :            - TargetValue[3] HW LB
// Byte 076 :            - TargetValue[3] LW HB
// Byte 077 :            - TargetValue[3] LW LB
// Byte 078 : REAL       - TargetValue[4] HW HB
// Byte 079 :            - TargetValue[4] HW LB
// Byte 080 :            - TargetValue[4] LW HB
// Byte 081 :            - TargetValue[4] LW LB
// Byte 082 : REAL       - TargetValue[5] HW HB
// Byte 083 :            - TargetValue[5] HW LB
// Byte 084 :            - TargetValue[5] LW HB
// Byte 085 :            - TargetValue[5] LW LB
// Byte 086 : UINT       - MaxVelocity LW HB
// Byte 087 :            - MaxVelocity LW LB
// Byte 088 : REAL       - MaxDeviation[0] HW HB
// Byte 089 :            - MaxDeviation[0] HW LB
// Byte 090 :            - MaxDeviation[0] LW HB
// Byte 091 :            - MaxDeviation[0] LW LB
// Byte 092 : REAL       - MaxDeviation[1] HW HB
// Byte 093 :            - MaxDeviation[1] HW LB
// Byte 094 :            - MaxDeviation[1] LW HB
// Byte 095 :            - MaxDeviation[1] LW LB
// Byte 096 : REAL       - MaxDeviation[2] HW HB
// Byte 097 :            - MaxDeviation[2] HW LB
// Byte 098 :            - MaxDeviation[2] LW HB
// Byte 099 :            - MaxDeviation[2] LW LB
// Byte 100 : REAL       - MaxDeviation[3] HW HB
// Byte 101 :            - MaxDeviation[3] HW LB
// Byte 102 :            - MaxDeviation[3] LW HB
// Byte 103 :            - MaxDeviation[3] LW LB
// Byte 104 : REAL       - MaxDeviation[4] HW HB
// Byte 105 :            - MaxDeviation[4] HW LB
// Byte 106 :            - MaxDeviation[4] LW HB
// Byte 107 :            - MaxDeviation[4] LW LB
// Byte 108 : REAL       - MaxDeviation[5] HW HB
// Byte 109 :            - MaxDeviation[5] HW LB
// Byte 110 :            - MaxDeviation[5] LW HB
// Byte 111 :            - MaxDeviation[5] LW LB
// Byte 112 : USINT      - ErrorReaction
// Byte 113 : USINT      - ErrorReferenceType
// Byte 114 : REAL       - ErrorVector[0] HW HB
// Byte 115 :            - ErrorVector[0] HW LB
// Byte 116 :            - ErrorVector[0] LW HB
// Byte 117 :            - ErrorVector[0] LW LB
// Byte 118 : REAL       - ErrorVector[1] HW HB
// Byte 119 :            - ErrorVector[1] HW LB
// Byte 120 :            - ErrorVector[1] LW HB
// Byte 121 :            - ErrorVector[1] LW LB
// Byte 122 : REAL       - ErrorVector[2] HW HB
// Byte 123 :            - ErrorVector[2] HW LB
// Byte 124 :            - ErrorVector[2] LW HB
// Byte 125 :            - ErrorVector[2] LW LB
// Byte 126 : REAL       - ErrorVector[3] HW HB
// Byte 127 :            - ErrorVector[3] HW LB
// Byte 128 :            - ErrorVector[3] LW HB
// Byte 129 :            - ErrorVector[3] LW LB
// Byte 130 : REAL       - ErrorVector[4] HW HB
// Byte 131 :            - ErrorVector[4] HW LB
// Byte 132 :            - ErrorVector[4] LW HB
// Byte 133 :            - ErrorVector[4] LW LB
// Byte 134 : REAL       - ErrorVector[5] HW HB
// Byte 135 :            - ErrorVector[5] HW LB
// Byte 136 :            - ErrorVector[5] LW HB
// Byte 137 :            - ErrorVector[5] LW LB
// Byte 138 : USINT      - ErrorToolNo
// Byte 139 : USINT      - ErrorFrameNo
// Byte 140 : BYTE       - CompliantAxes
// --------------------------
// set command parameter 
_command.CmdTyp             :=  CmdType.ForceControl;
_command.ExecMode           :=  ExecMode;
_command.ParSeq             := _command.ParSeq;
_command.Priority           :=  Priority;
_command.ToolNo             := _parCmd.ToolNo;
_command.FrameNo            := _parCmd.FrameNo;
_command.ConnectionMode     := _parCmd.ConnectionMode;
_command.FixedSensor.0      := _parCmd.FixedSensor;
_command.SensorFrame        := _parCmd.SensorFrame;
_command.CalibrationData    := _parCmd.CalibrationData;
_command.ReferenceType      := _parCmd.ReferenceType;
_command.SensorValue        := _parCmd.SensorValue;
_command.TargetValue        := _parCmd.TargetValue;
_command.MaxVelocity        := _parCmd.MaxVelocity;
_command.MaxDeviation       := _parCmd.MaxDeviation;
_command.ErrorReaction      := _parCmd.ErrorReaction;
_command.ErrorReferenceType := _parCmd.ErrorReferenceType;
_command.ErrorVector        := _parCmd.ErrorVector;
_command.ErrorToolNo        := _parCmd.ErrorToolNo;
_command.ErrorFrameNo       := _parCmd.ErrorFrameNo;
_command.CompliantAxes      := _parCmd.CompliantAxes;

// copy command data to header
_cmdHeader := _command;
// call base implementation to copy header to payload buffer
CreateCommandPayload := SUPER^.CreateCommandPayload(AxesGroup := AxesGroup);


